// TIA Portal project "VISU_F-Band+WzMaschine_Template" (V14)

(* hardware
DEVICE "S7300/ET200M-Station_1"  S7-300 station
   slot 0: "Profilschiene_0"  Rail  6ES7 390-1***0-0AA0
   slot 2: "PLC_1"  CPU 315-2 PN/DP  6ES7 315-2EH13-0AB0  V2.6
      slot 1: "MPI/DP-Schnittstelle_1"  X1
      slot 2: "PROFINET-Schnittstelle_1"  PN-IO
         slot 1: "Port_1"  Port
*)

// ===== PLC "PLC_1"  CPU 315-2 PN/DP =====

VAR_GLOBAL   // PLC tag table "Standard-Variablentabelle"
   "CONTROL_KEY" AT %I10.5 : Bool;   // Bedientaster
   "BELT_TO_X_PLUS" AT %Q4.0 : Bool;   // Förderband nach X+
   "BELT_ENGAGED" AT %I10.0 : Bool;   // Förderband belegt
   "POS_Y_PLUS" AT %I10.1 : Bool;   // Werkzeug bei Y+
   "POS_Y_MINUS" AT %I10.2 : Bool;   // Werkzeug bei Y-
   "POS_Z_PLUS" AT %I10.3 : Bool;   // Werkzeug bei Z+
   "POS_Z_MINUS" AT %I10.4 : Bool;   // Werkzeug bei Z-
   "TO_Y_PLUS" AT %Q4.2 : Bool;   // Werkzeug nach Y+
   "TO_Y_MINUS" AT %Q4.3 : Bool;   // Werkzeug nach Y-
   "TO_Z_PLUS" AT %Q4.4 : Bool;   // Werkzeug nach Z+
   "TO_Z_MINUS" AT %Q4.5 : Bool;   // Werkzeug nach Z-
   "TOOL_ON" AT %Q4.6 : Bool;   // Werkzeugantrieb
   "TIMER" AT %M1000.1 : Bool;   // Zeitgeber für Werkzeugantrieb
   "BELT_TO_X_MINUS" AT %Q4.1 : Bool;   // Förderband nach X-
   "WORKPIECE_STORE (FINISH)" AT %M1000.2 : Bool;   // Werkstückablage
   "INIT_1" AT %M0.2 : Bool;
   "INIT_0" AT %M0.1 : Bool;
   "STEP" AT %MW6 : Int;
   "MOVE_1" AT %M2.2 : Bool;
   "IN_CONSTRUCTION" AT %M0.3 : Bool;
   "TRIG_BELT_ENGANGED" AT %M0.7 : Bool;
   "MOVE_3" AT %M2.0 : Bool;
   "TRIG_Z_MINUS" AT %M1.0 : Bool;
   "TRIG_Y_MINUS" AT %M1.1 : Bool;
   "TRIG_Y_PLUS" AT %M1.2 : Bool;
   "TRIG_Z_PLUS" AT %M1.3 : Bool;
   "MOVE_2" AT %M2.1 : Bool;
   "TRIG_MOVE_NEG" AT %M1.6 : Bool;
   "TRIG_MOVE_POS" AT %M1.5 : Bool;
   "TRIG_BELT_ENGAGED_2" AT %M1.4 : Bool;
END_VAR

ORGANIZATION_BLOCK "Main"   // OB1, FBD
TITLE = "Main Program Sweep (Cycle)"
{ S7_Optimized_Access := 'FALSE' }
VERSION : 0.1
   VAR_TEMP
      OB1_EV_CLASS : Byte;   // Bits 0-3 = 1 (Coming event), Bits 4-7 = 1 (Event class 1)
      OB1_SCAN_1 : Byte;   // 1 (Cold restart scan 1 of OB 1), 3 (Scan 2-n of OB 1)
      OB1_PRIORITY : Byte;   // Priority of OB Execution
      OB1_OB_NUMBR : Byte;   // 1 (Organization block 1, OB1)
      OB1_RESERVED_1 : Byte;   // Reserved for system
      OB1_RESERVED_2 : Byte;   // Reserved for system
      OB1_PREV_CYCLE : Int;   // Cycle time of previous OB1 scan (milliseconds)
      OB1_MIN_CYCLE : Int;   // Minimum cycle time of OB1 (milliseconds)
      OB1_MAX_CYCLE : Int;   // Maximum cycle time of OB1 (milliseconds)
      OB1_DATE_TIME : Date_And_Time;   // Date and time OB1 started
   END_VAR
   VAR_TEMP   // added for the SCL form of the ladder/FBD networks
      _w1 : Bool;
      _w2 : Bool;
   END_VAR
BEGIN

REGION Network 1
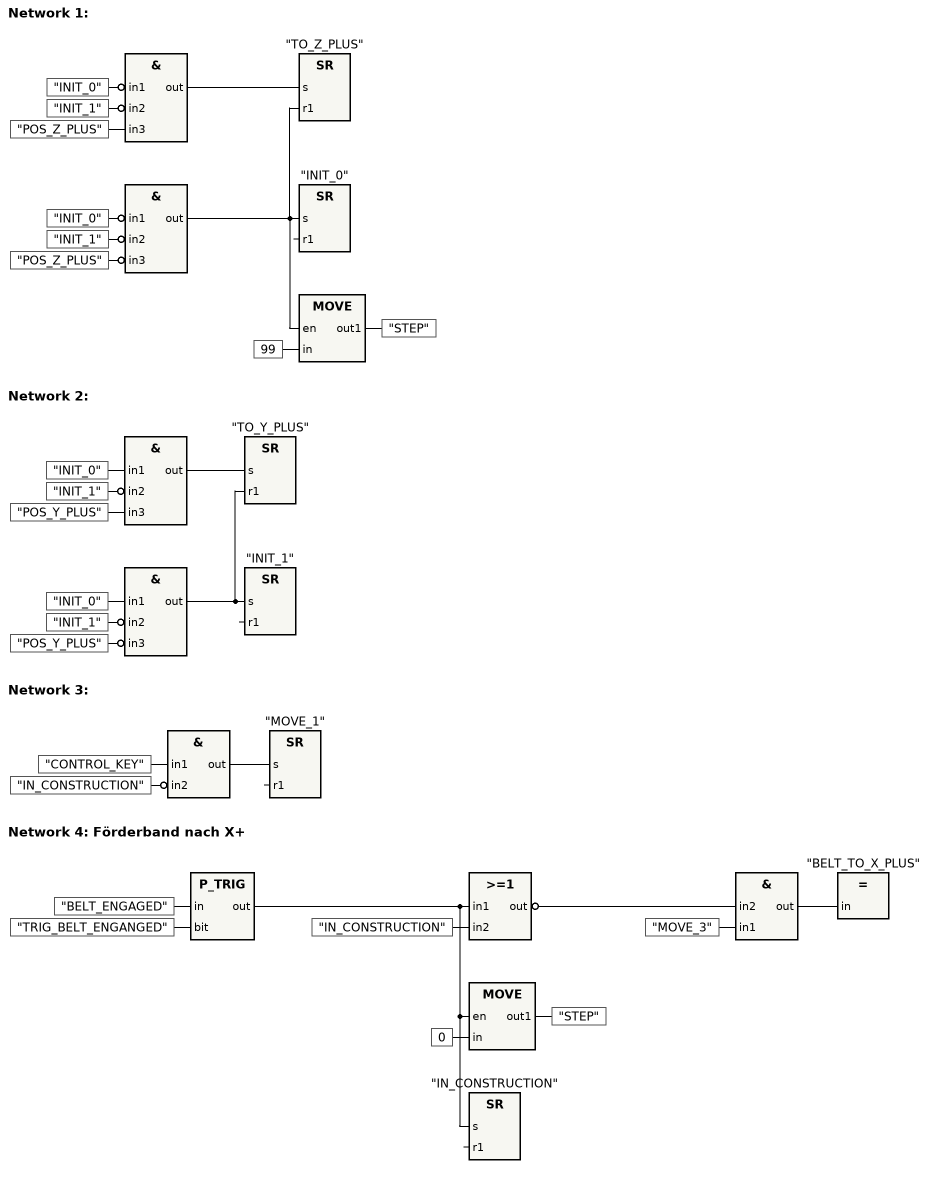
   #_w1 := NOT "INIT_0" AND NOT "INIT_1" AND NOT "POS_Z_PLUS";
   IF NOT "INIT_0" AND NOT "INIT_1" AND "POS_Z_PLUS" THEN
       "TO_Z_PLUS" := TRUE;   // SR flip-flop
   END_IF;
   IF #_w1 THEN
       "TO_Z_PLUS" := FALSE;
       "INIT_0" := TRUE;   // SR flip-flop
       "STEP" := 99;
   END_IF;
END_REGION

REGION Network 2
   #_w1 := "INIT_0" AND NOT "INIT_1" AND NOT "POS_Y_PLUS";
   IF "INIT_0" AND NOT "INIT_1" AND "POS_Y_PLUS" THEN
       "TO_Y_PLUS" := TRUE;   // SR flip-flop
   END_IF;
   IF #_w1 THEN
       "TO_Y_PLUS" := FALSE;
       "INIT_1" := TRUE;   // SR flip-flop
   END_IF;
END_REGION

REGION Network 3
   IF "CONTROL_KEY" AND NOT "IN_CONSTRUCTION" THEN
       "MOVE_1" := TRUE;   // SR flip-flop
   END_IF;
END_REGION

REGION Network 4: Förderband nach X+
   #_w1 := "BELT_ENGAGED" AND NOT "TRIG_BELT_ENGANGED";   // rising edge
   "TRIG_BELT_ENGANGED" := "BELT_ENGAGED";
   "BELT_TO_X_PLUS" := NOT (#_w1 OR "IN_CONSTRUCTION") AND "MOVE_3";
   IF #_w1 THEN
       "STEP" := 0;
       "IN_CONSTRUCTION" := TRUE;   // SR flip-flop
   END_IF;
END_REGION

REGION Network 5
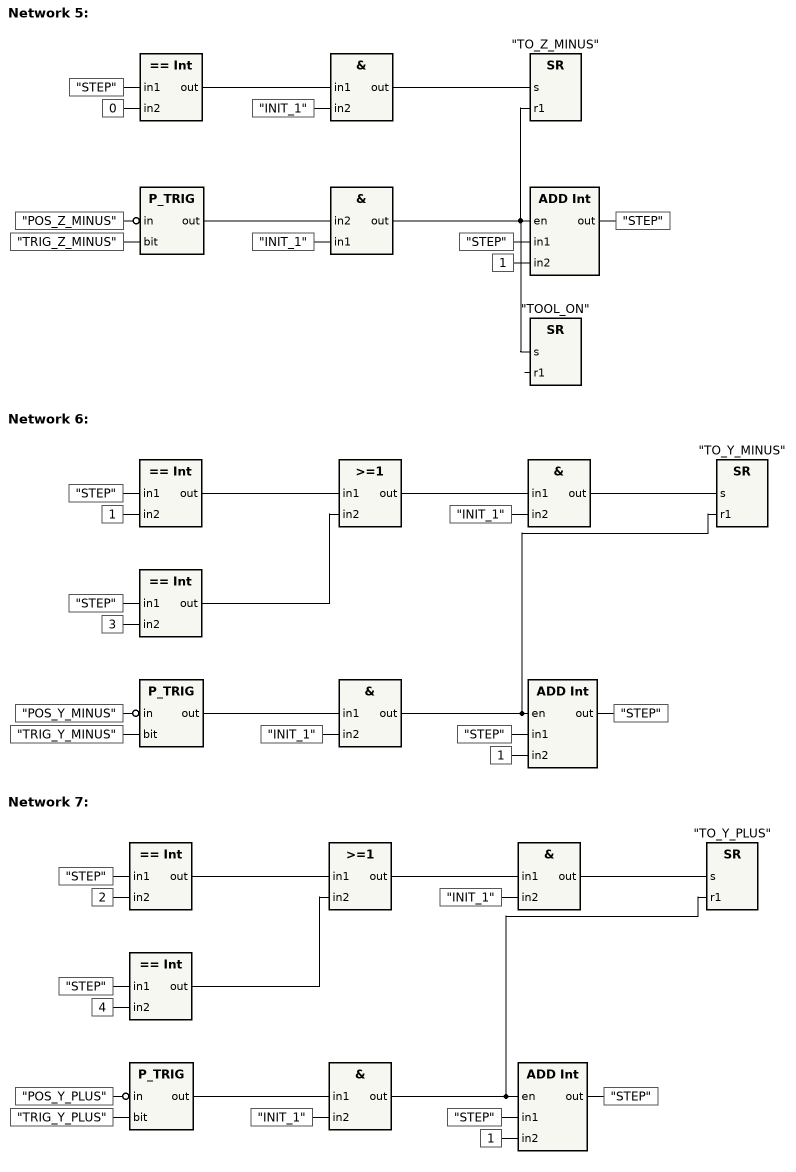
   #_w1 := NOT "POS_Z_MINUS" AND NOT "TRIG_Z_MINUS";   // rising edge
   "TRIG_Z_MINUS" := NOT "POS_Z_MINUS";
   #_w2 := #_w1 AND "INIT_1";
   IF ("STEP" = 0) AND "INIT_1" THEN
       "TO_Z_MINUS" := TRUE;   // SR flip-flop
   END_IF;
   IF #_w2 THEN
       "TO_Z_MINUS" := FALSE;
       "STEP" := "STEP" + 1;
       "TOOL_ON" := TRUE;   // SR flip-flop
   END_IF;
END_REGION

REGION Network 6
   #_w1 := NOT "POS_Y_MINUS" AND NOT "TRIG_Y_MINUS";   // rising edge
   "TRIG_Y_MINUS" := NOT "POS_Y_MINUS";
   #_w2 := #_w1 AND "INIT_1";
   IF (("STEP" = 1) OR ("STEP" = 3)) AND "INIT_1" THEN
       "TO_Y_MINUS" := TRUE;   // SR flip-flop
   END_IF;
   IF #_w2 THEN
       "TO_Y_MINUS" := FALSE;
       "STEP" := "STEP" + 1;
   END_IF;
END_REGION

REGION Network 7
   #_w1 := NOT "POS_Y_PLUS" AND NOT "TRIG_Y_PLUS";   // rising edge
   "TRIG_Y_PLUS" := NOT "POS_Y_PLUS";
   #_w2 := #_w1 AND "INIT_1";
   IF (("STEP" = 2) OR ("STEP" = 4)) AND "INIT_1" THEN
       "TO_Y_PLUS" := TRUE;   // SR flip-flop
   END_IF;
   IF #_w2 THEN
       "TO_Y_PLUS" := FALSE;
       "STEP" := "STEP" + 1;
   END_IF;
END_REGION

REGION Network 8
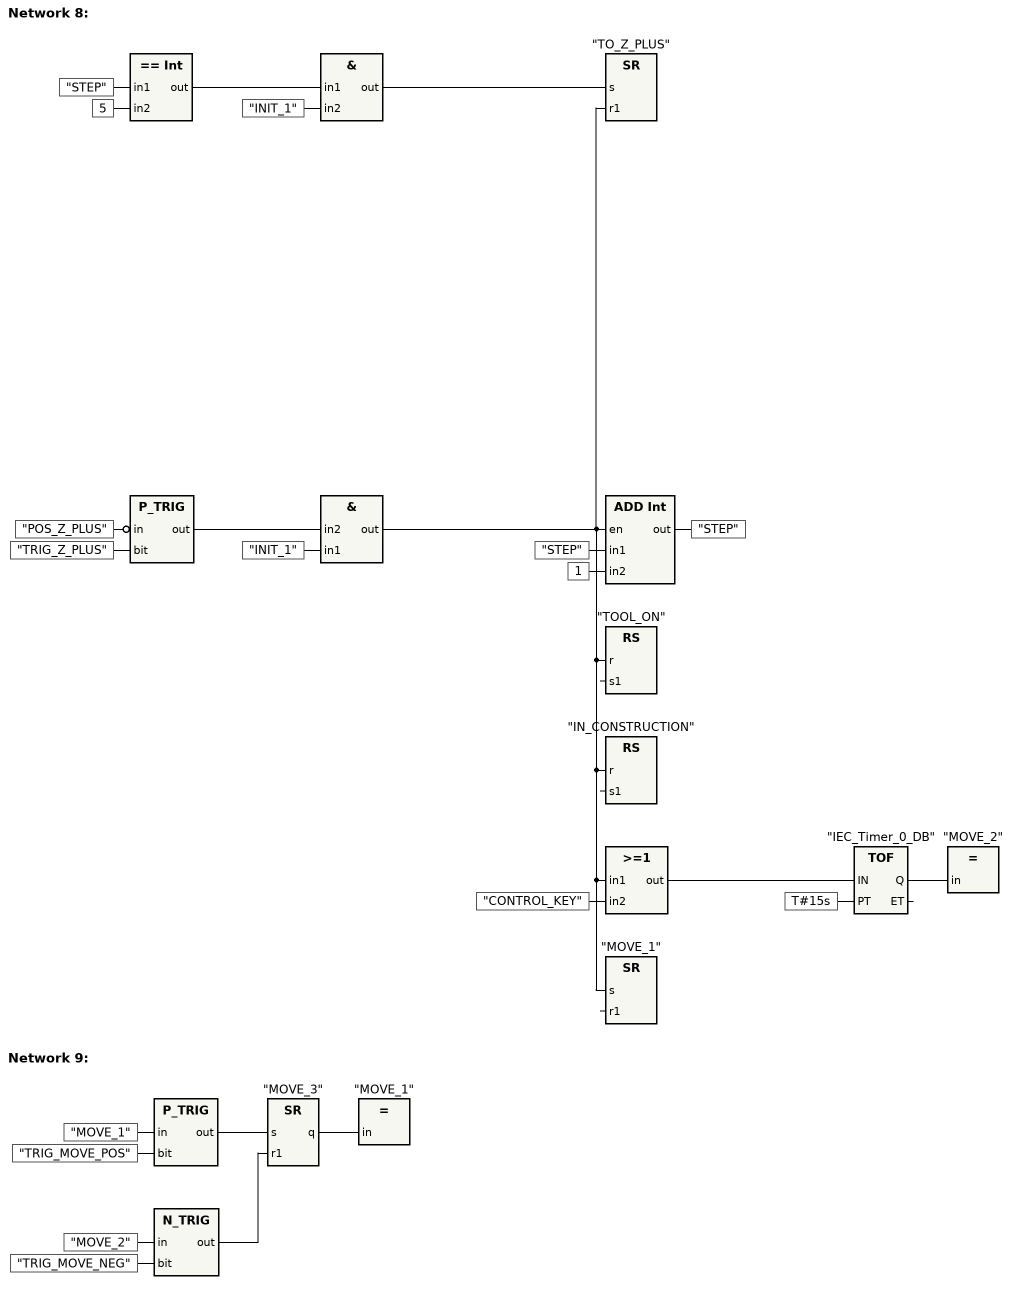
   #_w1 := NOT "POS_Z_PLUS" AND NOT "TRIG_Z_PLUS";   // rising edge
   "TRIG_Z_PLUS" := NOT "POS_Z_PLUS";
   #_w2 := #_w1 AND "INIT_1";
   IF ("STEP" = 5) AND "INIT_1" THEN
       "TO_Z_PLUS" := TRUE;   // SR flip-flop
   END_IF;
   IF #_w2 THEN
       "TO_Z_PLUS" := FALSE;
       "STEP" := "STEP" + 1;
       "TOOL_ON" := FALSE;   // RS flip-flop
       "IN_CONSTRUCTION" := FALSE;   // RS flip-flop
   END_IF;
   "IEC_Timer_0_DB".TOF(IN := #_w2 OR "CONTROL_KEY", PT := T#15s);
   "MOVE_2" := "IEC_Timer_0_DB".Q;
   IF #_w2 THEN
       "MOVE_1" := TRUE;   // SR flip-flop
   END_IF;
END_REGION

REGION Network 9
   #_w1 := "MOVE_1" AND NOT "TRIG_MOVE_POS";   // rising edge
   "TRIG_MOVE_POS" := "MOVE_1";
   #_w2 := NOT "MOVE_2" AND "TRIG_MOVE_NEG";   // falling edge
   "TRIG_MOVE_NEG" := "MOVE_2";
   IF #_w1 THEN
       "MOVE_3" := TRUE;   // SR flip-flop
   END_IF;
   IF #_w2 THEN "MOVE_3" := FALSE; END_IF;
   "MOVE_1" := "MOVE_3";
END_REGION

REGION Network 10
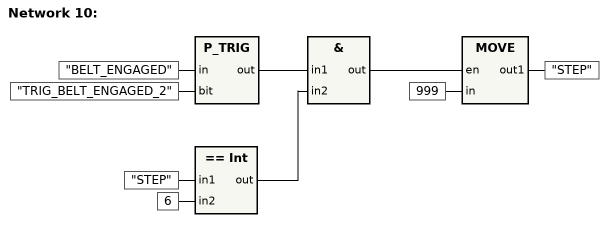
   #_w1 := "BELT_ENGAGED" AND NOT "TRIG_BELT_ENGAGED_2";   // rising edge
   "TRIG_BELT_ENGAGED_2" := "BELT_ENGAGED";
   IF #_w1 AND ("STEP" = 6) THEN "STEP" := 999; END_IF;
END_REGION
END_ORGANIZATION_BLOCK